INTERFACE I_HE_SATT_FilterHolder


METHOD GetConfiguration
VAR_OUTPUT
    stFilter : ARRAY[1..14] OF ST_Filter;
END_VAR
END_METHOD


METHOD GetFilter : ST_Filter
VAR_INPUT
    nFilterNumber : INT;
END_VAR
END_METHOD

PROPERTY NumberOfSlots : INT
GET
END_GET
END_PROPERTY

END_INTERFACE

(* stored: Version 1.1.0.1
   Itf I_HE_SATT_FilterHolder: Id {50894da0-cc33-47a4-8023-07412f59bfc3}
   Method GetConfiguration: Id {0dc13831-f14f-4407-90bf-710330175d68}
   Method GetFilter: Id {b9af26ac-850d-4c8d-8479-197f9f19bd28}
   Property NumberOfSlots: Id {e83b7fb5-7407-4813-b9cc-d270aebd7af9}
   Get Get: Id {3b73d66b-ce03-4755-bc84-99831ecd961a} *)
